TYPE ST_Cylinder :
STRUCT
	ExtendedCmd		: BOOL;
	RetractCmd		: BOOL;
	Extended		: BOOL;
END_STRUCT
END_TYPE

(* stored: Version 1.1.0.1, ProductVersion 3.1.4024.12
   DUT ST_Cylinder: Id {9909411d-711e-4020-9974-65a340bda058} *)
